PROGRAM prg_TweePompen
VAR
	Hoofdschakelaar			AT		%I*		:BOOL;
	StartKnop				AT		%I*		:BOOL;
	StopKnop				AT		%I*		:BOOL;
	NiveauSchakelaarOnder	AT		%I*		:BOOL;
	NiveauSchakelaarBoven	AT		%I*		:BOOL;
	
	Pomp1					AT		%Q*		:BOOL;
	Pomp2					AT		%Q*		:BOOL;
	PompWissel: BOOL;
	PompAan: BOOL;
	
END_VAR

IF Hoofdschakelaar AND (StartKnop OR NiveauSchakelaarOnder) AND NOT (StopKnop OR NiveauSchakelaarBoven) THEN
	PompAan:=TRUE;
ELSE
	PompAan:=False;	
END_IF

IF PompAan AND NOT Pomp1 AND NOT Pomp2 THEN
	PompWissel:= NOT PompWissel;
END_IF

IF PompAan THEN
    Pomp1 := PompWissel;
    Pomp2 := NOT PompWissel;
ELSE
    Pomp1 := FALSE;
    Pomp2 := FALSE;
END_IF

END_PROGRAM

(* stored: Version 1.1.0.1, ProductVersion 3.1.4024.15
   POU prg_TweePompen: Id {7048cf9a-ec8a-4d58-be81-622fef65ddd6}, SpecialFunc None *)
